{attribute 'qualified_only'}
{attribute 'strict'}
TYPE
    E_ClampAction :
    (
        Undefine := 0, // Clamp no action
        PickUp,        // Clamp catch something.
        Place          // Clamp release something.
    );
END_TYPE

(* stored: Version 1.1.0.1, ProductVersion 3.1.4024.13
   DUT E_ClampAction: Id {621609be-c15e-47e1-8c96-9858a7c79432} *)
